REGION Network 15: IO evaluation — Instrument read and scale - Part 2
   // ▀▀▀▀▀▀▀▀▀▀▀▀▀▀▀▀▀▀▀▀▀▀▀▀▀▀▀▀▀▀▀▀▀▀▀▀▀▀▀▀▀▀▀▀
   // Scale value calculation part 2 (SCALE_MAX − SCALE_MIN)
   // ▄▄▄▄▄▄▄▄▄▄▄▄▄▄▄▄▄▄▄▄▄▄▄▄▄▄▄▄▄▄▄▄▄▄▄▄▄▄▄▄▄▄▄▄
   RUNG wire#powerrail
      { S7_Templates := "SrcType := Real"; S7_GenerateENO := "TRUE" } Sub(in1 := #STATIC_DATA.RANGE_SCALE_MAX, in2 := #STATIC_DATA.RANGE_SCALE_MIN, out => #calcPart2)
   END_RUNG
   // the same network as SCL:
   #calcPart2 := #STATIC_DATA.RANGE_SCALE_MAX - #STATIC_DATA.RANGE_SCALE_MIN;
END_REGION

REGION Network 16: IO evaluation — Instrument read and scale - Part 3
   // ▀▀▀▀▀▀▀▀▀▀▀▀▀▀▀▀▀▀▀▀▀▀▀▀▀▀▀▀▀▀▀▀▀▀▀▀▀▀▀▀▀▀▀▀
   // Scale value calculation part 3 (RAW_MAX − RAW_MIN)
   // 
   // Note:    To prevent inconsistencies and divide by zero errors, if a configuration error is present
   //      (resulting from incorrect range data and indicated by status_ConfigError = TRUE), the
   //      denominator of the calculation (CalcPart3) is set to 3.402823 × 1038 (i.e. a very large 
   //      number), the result of this is that the  actual_Value will equal RANGE_SCALE_MIN for 
   //      all permitted values of RAW_ANALOG.
   // ▄▄▄▄▄▄▄▄▄▄▄▄▄▄▄▄▄▄▄▄▄▄▄▄▄▄▄▄▄▄▄▄▄▄▄▄▄▄▄▄▄▄▄▄
   RUNG wire#powerrail
      { S7_Templates := "SrcType := Real"; S7_GenerateENO := "TRUE" } Sub(in1 := #STATIC_DATA.RANGE_RAW_MAX, in2 := #STATIC_DATA.RANGE_RAW_MIN, out => #calcPart3)
      Contact( #DYNAMIC_DATA.status_ConfigError )
      Move(in := 3.402823E+38, out1 => #calcPart3)
   END_RUNG
   // the same network as SCL:
   // ENO of a box is taken as its EN; it also drops when the box reports an error
   #calcPart3 := #STATIC_DATA.RANGE_RAW_MAX - #STATIC_DATA.RANGE_RAW_MIN;
   IF #DYNAMIC_DATA.status_ConfigError THEN #calcPart3 := 3.402823E+38; END_IF;
END_REGION

REGION Network 17: IO evaluation — Instrument read and scale - Part 4
   // ▀▀▀▀▀▀▀▀▀▀▀▀▀▀▀▀▀▀▀▀▀▀▀▀▀▀▀▀▀▀▀▀▀▀▀▀▀▀▀▀▀▀▀▀
   //                                                                              (calcPart1 x CalcPart2)
   // Complete the calculation SCALE_VALUE =  —————————— + SCALE_MIN
   //                                                                                         calcPart3
   // 
   // If a configuration error exists, the actual value is set to zero for all conditions
   // ▄▄▄▄▄▄▄▄▄▄▄▄▄▄▄▄▄▄▄▄▄▄▄▄▄▄▄▄▄▄▄▄▄▄▄▄▄▄▄▄▄▄▄▄
   RUNG wire#powerrail
      { S7_Templates := "SrcType := Real"; S7_GenerateENO := "TRUE" } Mul(in1 := #calcPart1, in2 := #calcPart2, out => #wrkReal)
      { S7_Templates := "SrcType := Real"; S7_GenerateENO := "TRUE" } Div(in1 := #wrkReal, in2 := #calcPart3, out => #wrkReal)
      { S7_Templates := "SrcType := Real"; S7_GenerateENO := "TRUE" } Add(in1 := #wrkReal, in2 := #STATIC_DATA.RANGE_SCALE_MIN, out => #DYNAMIC_DATA.actual_Value)
   END_RUNG
   RUNG wire#powerrail
      Contact( #DYNAMIC_DATA.status_ConfigError )
      Move(in := 0.0, out1 => #DYNAMIC_DATA.actual_Value)
   END_RUNG
   // the same network as SCL:
   // ENO of a box is taken as its EN; it also drops when the box reports an error
   #wrkReal := #calcPart1 * #calcPart2;
   #wrkReal := #wrkReal / #calcPart3;
   #DYNAMIC_DATA.actual_Value := #wrkReal + #STATIC_DATA.RANGE_SCALE_MIN;
   IF #DYNAMIC_DATA.status_ConfigError THEN #DYNAMIC_DATA.actual_Value := 0.0; END_IF;
END_REGION

REGION Network 18: IO evaluation — Calculate out of range value
   // ▀▀▀▀▀▀▀▀▀▀▀▀▀▀▀▀▀▀▀▀▀▀▀▀▀▀▀▀▀▀▀▀▀▀▀▀▀▀▀▀▀▀▀▀
   // The out of range limits are calculated from the raw span of the instrument 
   // (RAW_MAX - RAW_MIN, stored in calcPart3).
   // 
   // The absolute value of the out of range tolerance is stored in calcRawOOR and is calculated as
   // follows:
   // 
   // 
   //                                (RAW_MAX - RAW_MIN) x wrkOORPercent
   // calcRawOOR  =  ————————————————————
   //                                                                100
   // 
   // OR
   // 
   //                               calcPart3 x wrkOORPercent
   // calcRawOOR  =  ——————————————
   //                                                 100
   // 
   // 
   // The instrument is over range if the RAW_ANALOG is greater than RAW_MAX + calcRawOOR
   // 
   // The instrument is under range if the RAW_ANALOG is less than RAW_MIN - calcRawOOR
   // ▄▄▄▄▄▄▄▄▄▄▄▄▄▄▄▄▄▄▄▄▄▄▄▄▄▄▄▄▄▄▄▄▄▄▄▄▄▄▄▄▄▄▄▄
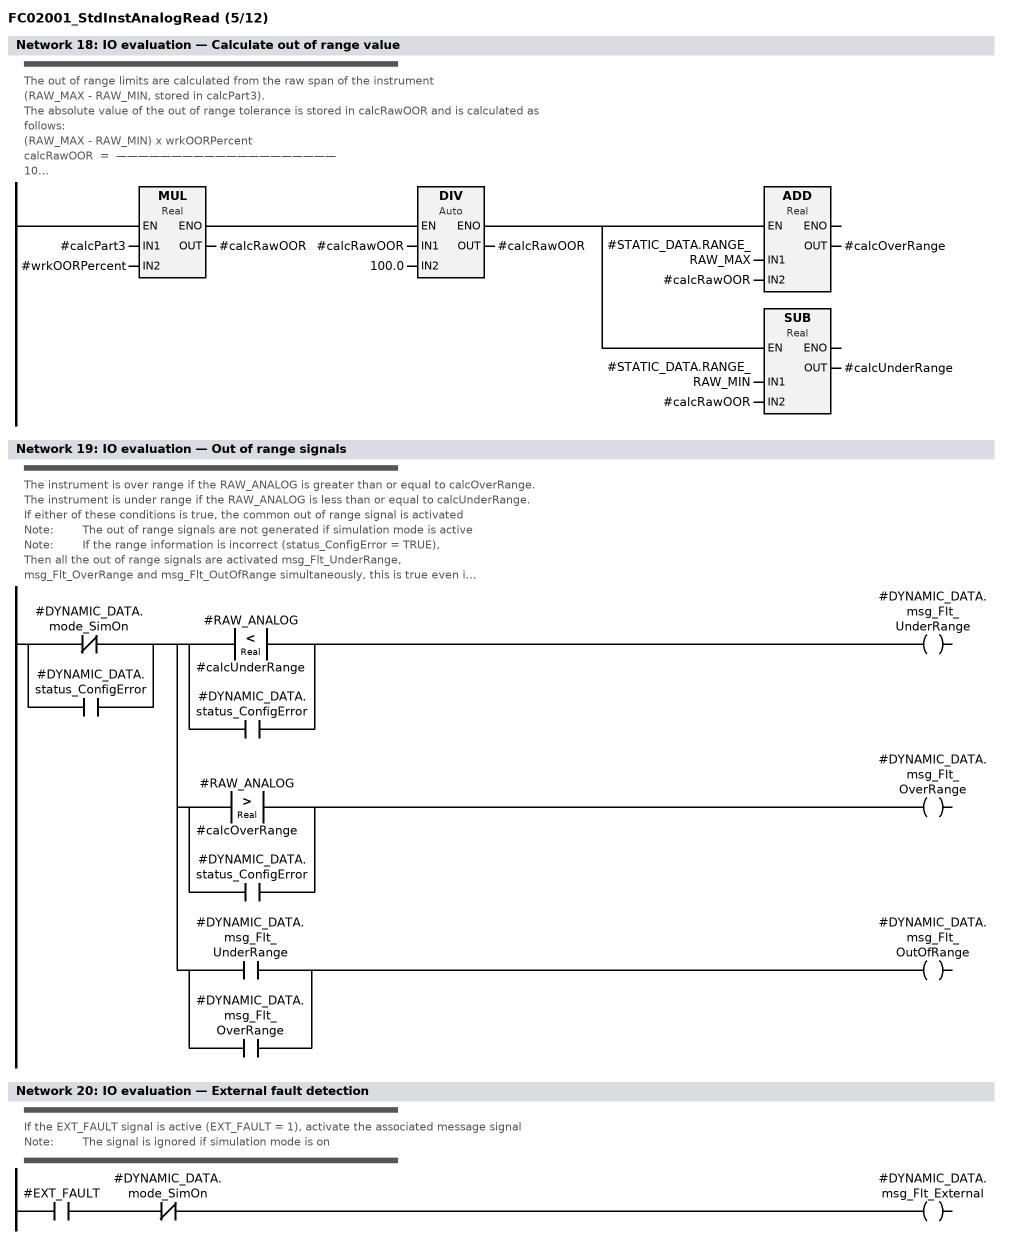
   RUNG wire#powerrail
      { S7_Templates := "SrcType := Real"; S7_GenerateENO := "TRUE" } Mul(in1 := #calcPart3, in2 := #wrkOORPercent, out => #calcRawOOR)
      Div(in1 := #calcRawOOR, in2 := 100.0, out => #calcRawOOR)
      wire#w1
      { S7_Templates := "SrcType := Real"; S7_GenerateENO := "TRUE" } Add(in1 := #STATIC_DATA.RANGE_RAW_MAX, in2 := #calcRawOOR, out => #calcOverRange)
   END_RUNG
   RUNG wire#w1
      { S7_Templates := "SrcType := Real"; S7_GenerateENO := "TRUE" } Sub(in1 := #STATIC_DATA.RANGE_RAW_MIN, in2 := #calcRawOOR, out => #calcUnderRange)
   END_RUNG
   // the same network as SCL:
   // ENO of a box is taken as its EN; it also drops when the box reports an error
   #calcRawOOR := #calcPart3 * #wrkOORPercent;
   #calcRawOOR := #calcRawOOR / 100.0;
   #calcOverRange := #STATIC_DATA.RANGE_RAW_MAX + #calcRawOOR;
   #calcUnderRange := #STATIC_DATA.RANGE_RAW_MIN - #calcRawOOR;
END_REGION

REGION Network 19: IO evaluation — Out of range signals
   // ▀▀▀▀▀▀▀▀▀▀▀▀▀▀▀▀▀▀▀▀▀▀▀▀▀▀▀▀▀▀▀▀▀▀▀▀▀▀▀▀▀▀▀▀
   // The instrument is over range if the RAW_ANALOG is greater than or equal to calcOverRange.
   // 
   // The instrument is under range if the RAW_ANALOG is less than or equal to calcUnderRange.
   // 
   // If either of these conditions is true, the common out of range signal is activated
   // 
   // Note:    The out of range signals are not generated if simulation mode is active
   // 
   // Note:    If the range information is incorrect (status_ConfigError = TRUE),
   //      Then all the out of range signals are activated msg_Flt_UnderRange, 
   //      msg_Flt_OverRange and msg_Flt_OutOfRange simultaneously, this is true even if
   //      simulation mode is active.
   // ▄▄▄▄▄▄▄▄▄▄▄▄▄▄▄▄▄▄▄▄▄▄▄▄▄▄▄▄▄▄▄▄▄▄▄▄▄▄▄▄▄▄▄▄
   RUNG wire#powerrail
      I_Contact( #DYNAMIC_DATA.mode_SimOn )
      wire#w1
      { S7_Templates := "SrcType := Real" } LT_Contact(in1 := #RAW_ANALOG, in2 := #calcUnderRange)
      wire#w2
      Coil( #DYNAMIC_DATA.msg_Flt_UnderRange )
   END_RUNG
   RUNG wire#powerrail
      Contact( #DYNAMIC_DATA.status_ConfigError )
   END_RUNG wire#w1
   RUNG wire#w1
      Contact( #DYNAMIC_DATA.status_ConfigError )
   END_RUNG wire#w2
   RUNG wire#w1
      { S7_Templates := "SrcType := Real" } GT_Contact(in1 := #RAW_ANALOG, in2 := #calcOverRange)
      wire#w3
      Coil( #DYNAMIC_DATA.msg_Flt_OverRange )
   END_RUNG
   RUNG wire#w1
      Contact( #DYNAMIC_DATA.status_ConfigError )
   END_RUNG wire#w3
   RUNG wire#w1
      Contact( #DYNAMIC_DATA.msg_Flt_UnderRange )
      wire#w4
      Coil( #DYNAMIC_DATA.msg_Flt_OutOfRange )
   END_RUNG
   RUNG wire#w1
      Contact( #DYNAMIC_DATA.msg_Flt_OverRange )
   END_RUNG wire#w4
   // the same network as SCL:
   #_w1 := NOT #DYNAMIC_DATA.mode_SimOn OR #DYNAMIC_DATA.status_ConfigError;
   #DYNAMIC_DATA.msg_Flt_UnderRange := #_w1 AND ((#RAW_ANALOG < #calcUnderRange) OR #DYNAMIC_DATA.status_ConfigError);
   #DYNAMIC_DATA.msg_Flt_OverRange := #_w1 AND ((#RAW_ANALOG > #calcOverRange) OR #DYNAMIC_DATA.status_ConfigError);
   #DYNAMIC_DATA.msg_Flt_OutOfRange := #_w1 AND (#DYNAMIC_DATA.msg_Flt_UnderRange OR #DYNAMIC_DATA.msg_Flt_OverRange);
END_REGION

REGION Network 20: IO evaluation — External fault detection
   // ▀▀▀▀▀▀▀▀▀▀▀▀▀▀▀▀▀▀▀▀▀▀▀▀▀▀▀▀▀▀▀▀▀▀▀▀▀▀▀▀▀▀▀▀
   // If the EXT_FAULT signal is active (EXT_FAULT = 1), activate the associated message signal
   // 
   // Note:    The signal is ignored if simulation mode is on
   // ▄▄▄▄▄▄▄▄▄▄▄▄▄▄▄▄▄▄▄▄▄▄▄▄▄▄▄▄▄▄▄▄▄▄▄▄▄▄▄▄▄▄▄▄
   RUNG wire#powerrail
      Contact( #EXT_FAULT )
      I_Contact( #DYNAMIC_DATA.mode_SimOn )
      Coil( #DYNAMIC_DATA.msg_Flt_External )
   END_RUNG
   // the same network as SCL:
   #DYNAMIC_DATA.msg_Flt_External := #EXT_FAULT AND NOT #DYNAMIC_DATA.mode_SimOn;
END_REGION

REGION Network 21: Operating mode — Simulation mode
   // ▀▀▀▀▀▀▀▀▀▀▀▀▀▀▀▀▀▀▀▀▀▀▀▀▀▀▀▀▀▀▀▀▀▀▀▀▀▀▀▀▀▀▀▀
   // If simulation mode is enabled (mode_SimOn = 1) and a configuration error is not present,
   // (status_ConfigError = 0) overwrite the actual_Value with the mode_SimValue signal set by the 
   // operator.
   // 
   // Note:    Any fault signals will be suppressed (turned off) is simulation mode is active
   //      and a configuration error is not present
   // 
   //      The simulated value (mode_SimValue) is restricted to the range given in 
   //      RANGE_SCALE_MIN and RANGE_SCALE_MAX
   // ▄▄▄▄▄▄▄▄▄▄▄▄▄▄▄▄▄▄▄▄▄▄▄▄▄▄▄▄▄▄▄▄▄▄▄▄▄▄▄▄▄▄▄▄
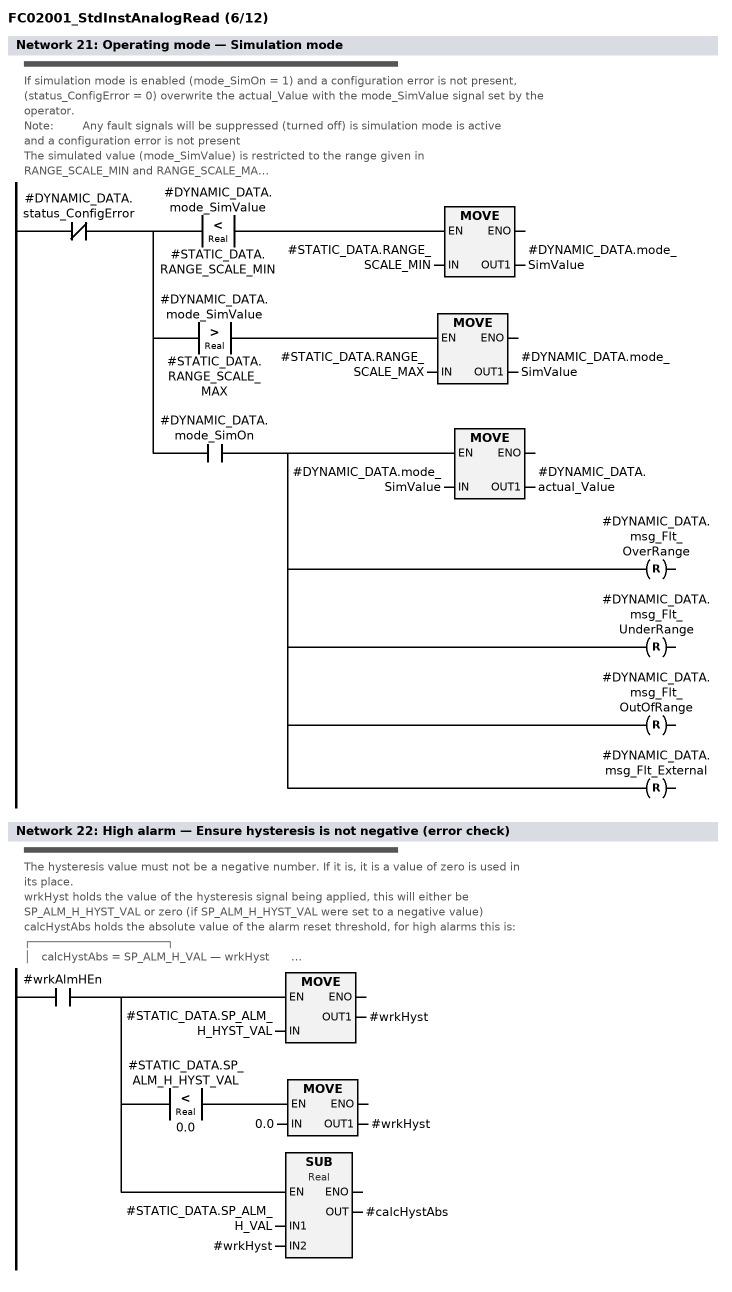
   RUNG wire#powerrail
      I_Contact( #DYNAMIC_DATA.status_ConfigError )
      wire#w1
      { S7_Templates := "SrcType := Real" } LT_Contact(in1 := #DYNAMIC_DATA.mode_SimValue, in2 := #STATIC_DATA.RANGE_SCALE_MIN)
      { S7_GenerateENO := "TRUE" } Move(in := #STATIC_DATA.RANGE_SCALE_MIN, out1 => #DYNAMIC_DATA.mode_SimValue)
   END_RUNG
   RUNG wire#w1
      { S7_Templates := "SrcType := Real" } GT_Contact(in1 := #DYNAMIC_DATA.mode_SimValue, in2 := #STATIC_DATA.RANGE_SCALE_MAX)
      { S7_GenerateENO := "TRUE" } Move(in := #STATIC_DATA.RANGE_SCALE_MAX, out1 => #DYNAMIC_DATA.mode_SimValue)
   END_RUNG
   RUNG wire#w1
      Contact( #DYNAMIC_DATA.mode_SimOn )
      wire#w2
      { S7_GenerateENO := "TRUE" } Move(in := #DYNAMIC_DATA.mode_SimValue, out1 => #DYNAMIC_DATA.actual_Value)
   END_RUNG
   RUNG wire#w2
      R_Coil( #DYNAMIC_DATA.msg_Flt_OverRange )
   END_RUNG
   RUNG wire#w2
      R_Coil( #DYNAMIC_DATA.msg_Flt_UnderRange )
   END_RUNG
   RUNG wire#w2
      R_Coil( #DYNAMIC_DATA.msg_Flt_OutOfRange )
   END_RUNG
   RUNG wire#w2
      R_Coil( #DYNAMIC_DATA.msg_Flt_External )
   END_RUNG
   // the same network as SCL:
   #_w1 := NOT #DYNAMIC_DATA.status_ConfigError;
   IF #_w1 AND (#DYNAMIC_DATA.mode_SimValue < #STATIC_DATA.RANGE_SCALE_MIN) THEN
       #DYNAMIC_DATA.mode_SimValue := #STATIC_DATA.RANGE_SCALE_MIN;
   END_IF;
   IF #_w1 AND (#DYNAMIC_DATA.mode_SimValue > #STATIC_DATA.RANGE_SCALE_MAX) THEN
       #DYNAMIC_DATA.mode_SimValue := #STATIC_DATA.RANGE_SCALE_MAX;
   END_IF;
   IF #_w1 AND #DYNAMIC_DATA.mode_SimOn THEN
       #DYNAMIC_DATA.actual_Value := #DYNAMIC_DATA.mode_SimValue;
       #DYNAMIC_DATA.msg_Flt_OverRange := FALSE;
       #DYNAMIC_DATA.msg_Flt_UnderRange := FALSE;
       #DYNAMIC_DATA.msg_Flt_OutOfRange := FALSE;
       #DYNAMIC_DATA.msg_Flt_External := FALSE;
   END_IF;
END_REGION

REGION Network 22: High alarm — Ensure hysteresis is not negative (error check)
   // ▀▀▀▀▀▀▀▀▀▀▀▀▀▀▀▀▀▀▀▀▀▀▀▀▀▀▀▀▀▀▀▀▀▀▀▀▀▀▀▀▀▀▀▀
   // The hysteresis value must not be a negative number. If it is, it is a value of zero is used in
   // its place.
   // 
   // wrkHyst holds the value of the hysteresis signal being applied, this will either be 
   // SP_ALM_H_HYST_VAL or zero (if SP_ALM_H_HYST_VAL were set to a negative value)
   // 
   // calcHystAbs holds the absolute value of the alarm reset threshold, for high alarms this is:
   // ┌─────────────────────┐
   // │ calcHystAbs = SP_ALM_H_VAL — wrkHyst    │
   // └─────────────────────┘
   // 
   // The two threshold values for the high alarm are thus:
   // 
   //      High alarm activation threshold = SP_ALM_H_VAL
   //      High alarm reset threshold          = calcHystAbs
   // 
   // Note:    The hysteresis is only checked if alarm is being evaluated
   // ▄▄▄▄▄▄▄▄▄▄▄▄▄▄▄▄▄▄▄▄▄▄▄▄▄▄▄▄▄▄▄▄▄▄▄▄▄▄▄▄▄▄▄▄
   RUNG wire#powerrail
      Contact( #wrkAlmHEn )
      wire#w1
      { S7_GenerateENO := "TRUE" } Move(in := #STATIC_DATA.SP_ALM_H_HYST_VAL, out1 => #wrkHyst)
   END_RUNG
   RUNG wire#w1
      { S7_Templates := "SrcType := Real" } LT_Contact(in1 := #STATIC_DATA.SP_ALM_H_HYST_VAL, in2 := 0.0)
      { S7_GenerateENO := "TRUE" } Move(in := 0.0, out1 => #wrkHyst)
   END_RUNG
   RUNG wire#w1
      { S7_Templates := "SrcType := Real"; S7_GenerateENO := "TRUE" } Sub(in1 := #STATIC_DATA.SP_ALM_H_VAL, in2 := #wrkHyst, out => #calcHystAbs)
   END_RUNG
   // the same network as SCL:
   IF #wrkAlmHEn THEN #wrkHyst := #STATIC_DATA.SP_ALM_H_HYST_VAL; END_IF;
   IF #wrkAlmHEn AND (#STATIC_DATA.SP_ALM_H_HYST_VAL < 0.0) THEN #wrkHyst := 0.0; END_IF;
   IF #wrkAlmHEn THEN #calcHystAbs := #STATIC_DATA.SP_ALM_H_VAL - #wrkHyst; END_IF;
END_REGION

REGION Network 23: High alarm — Check for activation level and ON-DELAY timer
   // ▀▀▀▀▀▀▀▀▀▀▀▀▀▀▀▀▀▀▀▀▀▀▀▀▀▀▀▀▀▀▀▀▀▀▀▀▀▀▀▀▀▀▀▀
   // If the high alarm has been enabled and is not masked and the actual_Value is greater than or 
   // equal to the alarm setpoint (SP_ALM_H_VAL), but the alarm has not yet been triggered 
   // (msg_Alm_H = 0) then the ON-DELAY phase is active (the alarm timer is counting down).
   // 
   // The timer will begin to count down from the value in TIME_ALM_H_ON_DEL using the 200ms 
   // pulse (it will count down in increments of 0.2s). If the high alarm timer is less than or equal to 
   // zero, then the ON-DELAY has expired and the High Alarm message will become active.
   // 
   // If at any point during the ON-DELAY count down, the actual_Value drops below the activation
   // setpoint (SP_ALM_H_VAL), the timer will be reset to the TIME_ALM_H_ON_DEL value, forcing 
   // the ON-DELAY to start again.
   // ▄▄▄▄▄▄▄▄▄▄▄▄▄▄▄▄▄▄▄▄▄▄▄▄▄▄▄▄▄▄▄▄▄▄▄▄▄▄▄▄▄▄▄▄
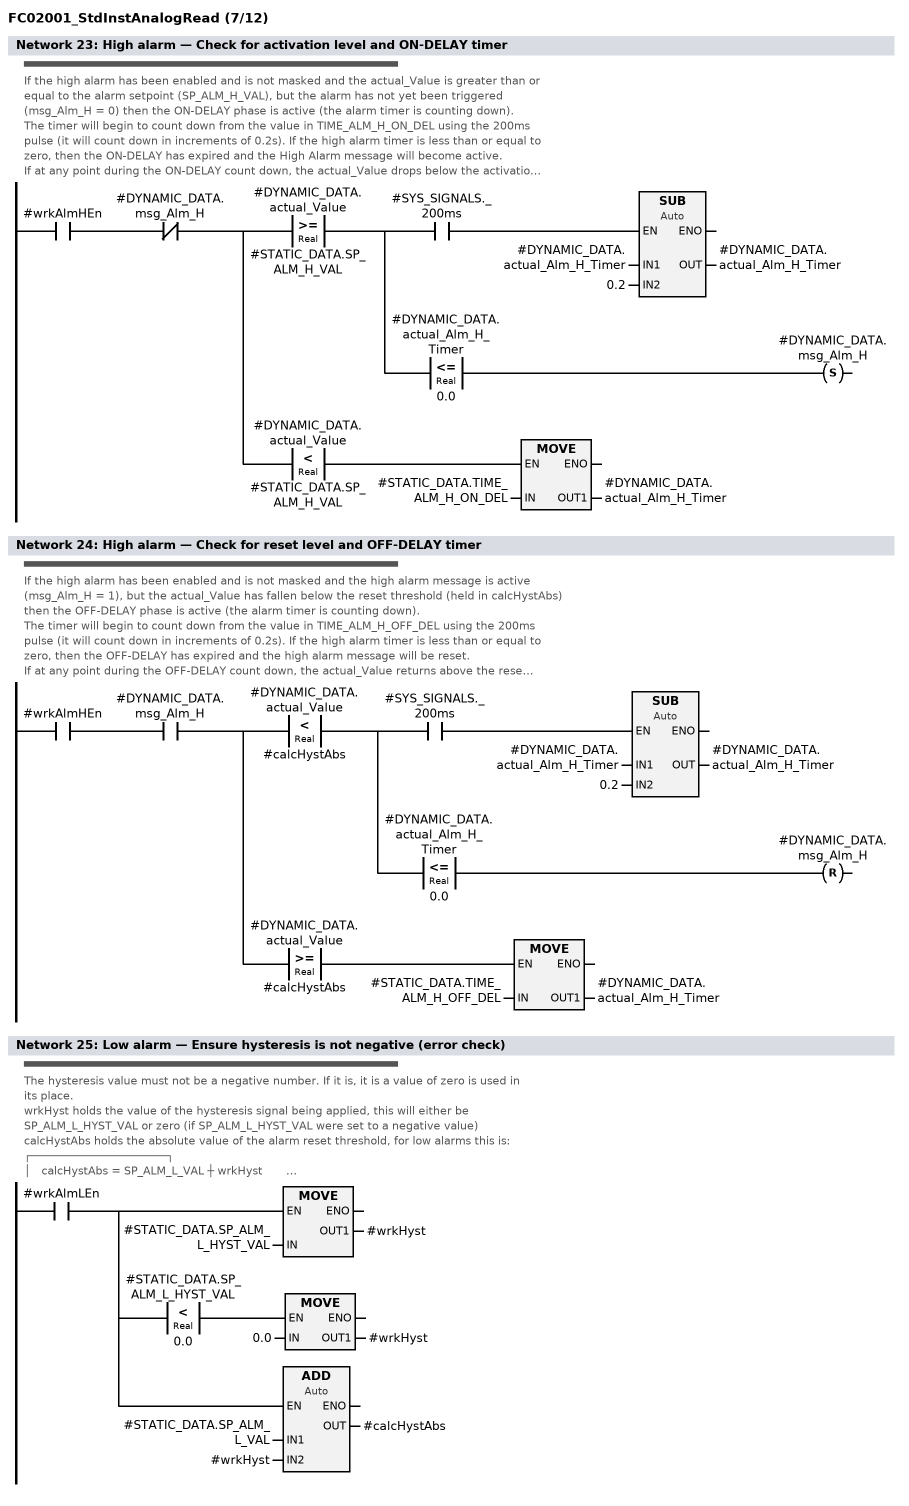
   RUNG wire#powerrail
      Contact( #wrkAlmHEn )
      I_Contact( #DYNAMIC_DATA.msg_Alm_H )
      wire#w1
      { S7_Templates := "SrcType := Real" } GE_Contact(in1 := #DYNAMIC_DATA.actual_Value, in2 := #STATIC_DATA.SP_ALM_H_VAL)
      wire#w2
      Contact( #SYS_SIGNALS._200ms )
      Sub(in1 := #DYNAMIC_DATA.actual_Alm_H_Timer, in2 := 0.2, out => #DYNAMIC_DATA.actual_Alm_H_Timer)
   END_RUNG
   RUNG wire#w2
      { S7_Templates := "SrcType := Real" } LE_Contact(in1 := #DYNAMIC_DATA.actual_Alm_H_Timer, in2 := 0.0)
      S_Coil( #DYNAMIC_DATA.msg_Alm_H )
   END_RUNG
   RUNG wire#w1
      { S7_Templates := "SrcType := Real" } LT_Contact(in1 := #DYNAMIC_DATA.actual_Value, in2 := #STATIC_DATA.SP_ALM_H_VAL)
      { S7_GenerateENO := "TRUE" } Move(in := #STATIC_DATA.TIME_ALM_H_ON_DEL, out1 => #DYNAMIC_DATA.actual_Alm_H_Timer)
   END_RUNG
   // the same network as SCL:
   #_w1 := #wrkAlmHEn AND NOT #DYNAMIC_DATA.msg_Alm_H;
   #_w2 := #_w1 AND (#DYNAMIC_DATA.actual_Value >= #STATIC_DATA.SP_ALM_H_VAL);
   IF #_w2 AND #SYS_SIGNALS._200ms THEN
       #DYNAMIC_DATA.actual_Alm_H_Timer := #DYNAMIC_DATA.actual_Alm_H_Timer - 0.2;
   END_IF;
   IF #_w2 AND (#DYNAMIC_DATA.actual_Alm_H_Timer <= 0.0) THEN #DYNAMIC_DATA.msg_Alm_H := TRUE; END_IF;
   IF #_w1 AND (#DYNAMIC_DATA.actual_Value < #STATIC_DATA.SP_ALM_H_VAL) THEN
       #DYNAMIC_DATA.actual_Alm_H_Timer := #STATIC_DATA.TIME_ALM_H_ON_DEL;
   END_IF;
END_REGION

REGION Network 24: High alarm — Check for reset level and OFF-DELAY timer
   // ▀▀▀▀▀▀▀▀▀▀▀▀▀▀▀▀▀▀▀▀▀▀▀▀▀▀▀▀▀▀▀▀▀▀▀▀▀▀▀▀▀▀▀▀
   // If the high alarm has been enabled and is not masked and the high alarm message is active 
   // (msg_Alm_H = 1), but the actual_Value has fallen below the reset threshold (held in calcHystAbs) 
   // then the OFF-DELAY phase is active (the alarm timer is counting down).
   // 
   // The timer will begin to count down from the value in TIME_ALM_H_OFF_DEL using the 200ms 
   // pulse (it will count down in increments of 0.2s). If the high alarm timer is less than or equal to 
   // zero, then the OFF-DELAY has expired and the high alarm message will be reset.
   // 
   // If at any point during the OFF-DELAY count down, the actual_Value returns above the reset
   // threshold (calcHystAbs), the timer will be reset to the TIME_ALM_H_OFF_DEL value, forcing 
   // the OFF-DELAY to start again.
   // ▄▄▄▄▄▄▄▄▄▄▄▄▄▄▄▄▄▄▄▄▄▄▄▄▄▄▄▄▄▄▄▄▄▄▄▄▄▄▄▄▄▄▄▄
   RUNG wire#powerrail
      Contact( #wrkAlmHEn )
      Contact( #DYNAMIC_DATA.msg_Alm_H )
      wire#w1
      { S7_Templates := "SrcType := Real" } LT_Contact(in1 := #DYNAMIC_DATA.actual_Value, in2 := #calcHystAbs)
      wire#w2
      Contact( #SYS_SIGNALS._200ms )
      Sub(in1 := #DYNAMIC_DATA.actual_Alm_H_Timer, in2 := 0.2, out => #DYNAMIC_DATA.actual_Alm_H_Timer)
   END_RUNG
   RUNG wire#w2
      { S7_Templates := "SrcType := Real" } LE_Contact(in1 := #DYNAMIC_DATA.actual_Alm_H_Timer, in2 := 0.0)
      R_Coil( #DYNAMIC_DATA.msg_Alm_H )
   END_RUNG
   RUNG wire#w1
      { S7_Templates := "SrcType := Real" } GE_Contact(in1 := #DYNAMIC_DATA.actual_Value, in2 := #calcHystAbs)
      { S7_GenerateENO := "TRUE" } Move(in := #STATIC_DATA.TIME_ALM_H_OFF_DEL, out1 => #DYNAMIC_DATA.actual_Alm_H_Timer)
   END_RUNG
   // the same network as SCL:
   #_w1 := #wrkAlmHEn AND #DYNAMIC_DATA.msg_Alm_H;
   #_w2 := #_w1 AND (#DYNAMIC_DATA.actual_Value < #calcHystAbs);
   IF #_w2 AND #SYS_SIGNALS._200ms THEN
       #DYNAMIC_DATA.actual_Alm_H_Timer := #DYNAMIC_DATA.actual_Alm_H_Timer - 0.2;
   END_IF;
   IF #_w2 AND (#DYNAMIC_DATA.actual_Alm_H_Timer <= 0.0) THEN #DYNAMIC_DATA.msg_Alm_H := FALSE; END_IF;
   IF #_w1 AND (#DYNAMIC_DATA.actual_Value >= #calcHystAbs) THEN
       #DYNAMIC_DATA.actual_Alm_H_Timer := #STATIC_DATA.TIME_ALM_H_OFF_DEL;
   END_IF;
END_REGION

REGION Network 25: Low alarm — Ensure hysteresis is not negative (error check)
   // ▀▀▀▀▀▀▀▀▀▀▀▀▀▀▀▀▀▀▀▀▀▀▀▀▀▀▀▀▀▀▀▀▀▀▀▀▀▀▀▀▀▀▀▀
   // The hysteresis value must not be a negative number. If it is, it is a value of zero is used in
   // its place.
   // 
   // wrkHyst holds the value of the hysteresis signal being applied, this will either be 
   // SP_ALM_L_HYST_VAL or zero (if SP_ALM_L_HYST_VAL were set to a negative value)
   // 
   // calcHystAbs holds the absolute value of the alarm reset threshold, for low alarms this is:
   // ┌─────────────────────┐
   // │ calcHystAbs = SP_ALM_L_VAL ┼ wrkHyst     │
   // └─────────────────────┘
   // 
   // The two threshold values for the low alarm are thus:
   // 
   //      Low alarm activation threshold = SP_ALM_L_VAL
   //      Low alarm reset threshold          = calcHystAbs
   // 
   // Note:    The hysteresis is only checked if alarm is being evaluated
   // ▄▄▄▄▄▄▄▄▄▄▄▄▄▄▄▄▄▄▄▄▄▄▄▄▄▄▄▄▄▄▄▄▄▄▄▄▄▄▄▄▄▄▄▄
   RUNG wire#powerrail
      Contact( #wrkAlmLEn )
      wire#w1
      { S7_GenerateENO := "TRUE" } Move(in := #STATIC_DATA.SP_ALM_L_HYST_VAL, out1 => #wrkHyst)
   END_RUNG
   RUNG wire#w1
      { S7_Templates := "SrcType := Real" } LT_Contact(in1 := #STATIC_DATA.SP_ALM_L_HYST_VAL, in2 := 0.0)
      { S7_GenerateENO := "TRUE" } Move(in := 0.0, out1 => #wrkHyst)
   END_RUNG
   RUNG wire#w1
      Add(in1 := #STATIC_DATA.SP_ALM_L_VAL, in2 := #wrkHyst, out => #calcHystAbs)
   END_RUNG
   // the same network as SCL:
   IF #wrkAlmLEn THEN #wrkHyst := #STATIC_DATA.SP_ALM_L_HYST_VAL; END_IF;
   IF #wrkAlmLEn AND (#STATIC_DATA.SP_ALM_L_HYST_VAL < 0.0) THEN #wrkHyst := 0.0; END_IF;
   IF #wrkAlmLEn THEN #calcHystAbs := #STATIC_DATA.SP_ALM_L_VAL + #wrkHyst; END_IF;
END_REGION

REGION Network 26: Low alarm — Check for activation level and ON-DELAY timer
   // ▀▀▀▀▀▀▀▀▀▀▀▀▀▀▀▀▀▀▀▀▀▀▀▀▀▀▀▀▀▀▀▀▀▀▀▀▀▀▀▀▀▀▀▀
   // If the low alarm has been enabled and is not masked and the actual_Value is less than or 
   // equal to the alarm setpoint (SP_ALM_L_VAL), but the alarm has not yet been triggered 
   // (msg_Alm_L = 0) then the ON-DELAY phase is active (the alarm timer is counting down).
   // 
   // The timer will begin to count down from the value in TIME_ALM_L_ON_DEL using the 200ms 
   // pulse (it will count down in increments of 0.2s). If the Low alarm timer is less than or equal to 
   // zero, then the ON-DELAY has expired and the Low Alarm message will become active.
   // 
   // If at any point during the ON-DELAY count down, the actual_Value rises above the activation
   // setpoint (SP_ALM_L_VAL), the timer will be reset to the TIME_ALM_L_ON_DEL value, forcing 
   // the ON-DELAY to start again.
   // ▄▄▄▄▄▄▄▄▄▄▄▄▄▄▄▄▄▄▄▄▄▄▄▄▄▄▄▄▄▄▄▄▄▄▄▄▄▄▄▄▄▄▄▄
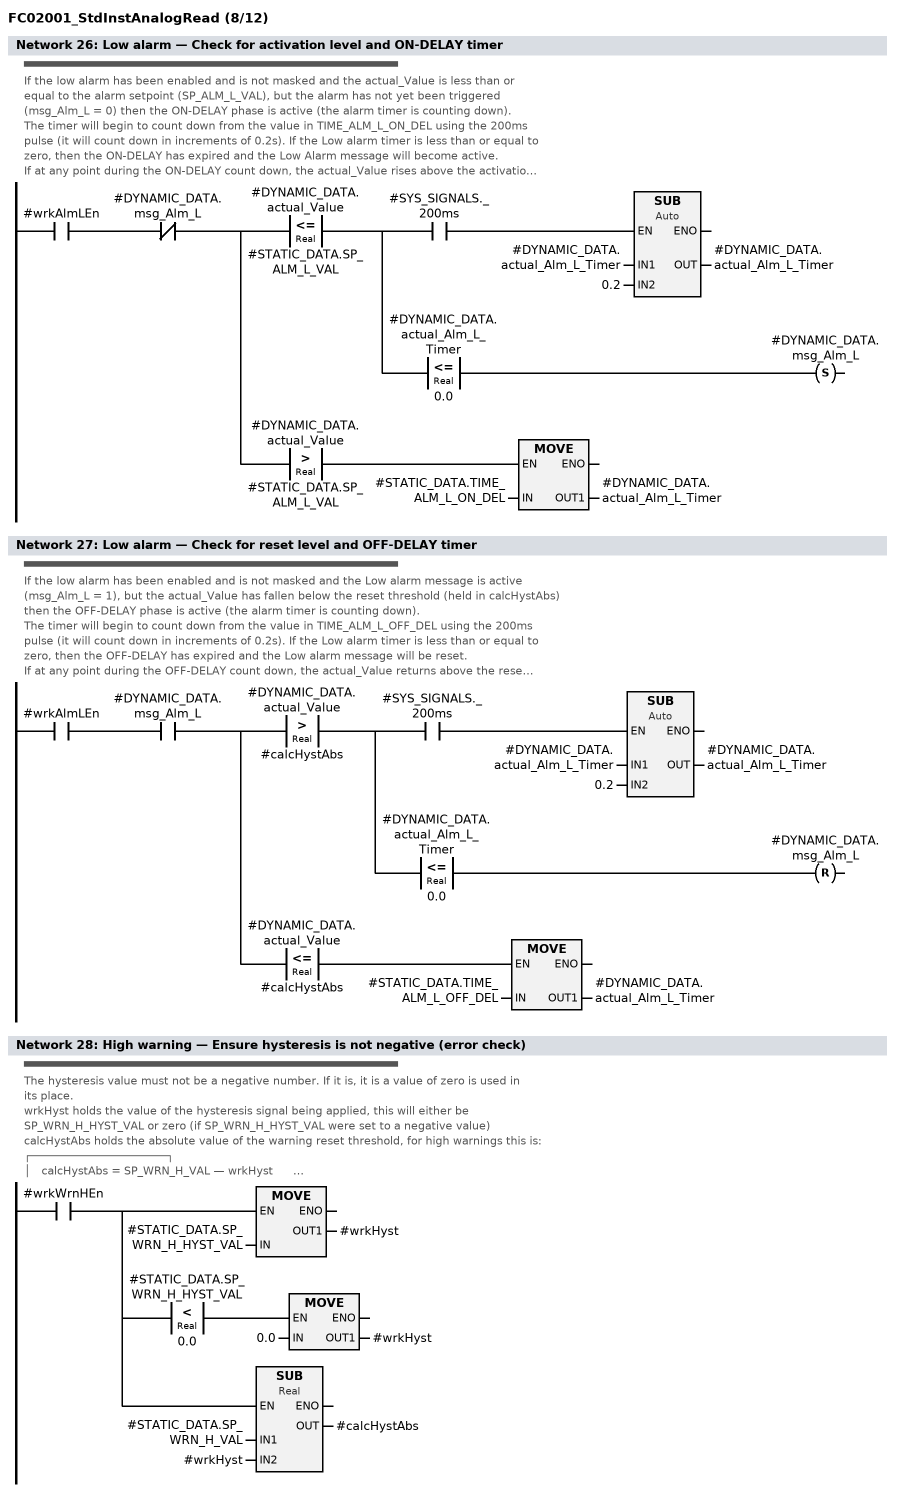
   RUNG wire#powerrail
      Contact( #wrkAlmLEn )
      I_Contact( #DYNAMIC_DATA.msg_Alm_L )
      wire#w1
      { S7_Templates := "SrcType := Real" } LE_Contact(in1 := #DYNAMIC_DATA.actual_Value, in2 := #STATIC_DATA.SP_ALM_L_VAL)
      wire#w2
      Contact( #SYS_SIGNALS._200ms )
      Sub(in1 := #DYNAMIC_DATA.actual_Alm_L_Timer, in2 := 0.2, out => #DYNAMIC_DATA.actual_Alm_L_Timer)
   END_RUNG
   RUNG wire#w2
      { S7_Templates := "SrcType := Real" } LE_Contact(in1 := #DYNAMIC_DATA.actual_Alm_L_Timer, in2 := 0.0)
      S_Coil( #DYNAMIC_DATA.msg_Alm_L )
   END_RUNG
   RUNG wire#w1
      { S7_Templates := "SrcType := Real" } GT_Contact(in1 := #DYNAMIC_DATA.actual_Value, in2 := #STATIC_DATA.SP_ALM_L_VAL)
      { S7_GenerateENO := "TRUE" } Move(in := #STATIC_DATA.TIME_ALM_L_ON_DEL, out1 => #DYNAMIC_DATA.actual_Alm_L_Timer)
   END_RUNG
   // the same network as SCL:
   #_w1 := #wrkAlmLEn AND NOT #DYNAMIC_DATA.msg_Alm_L;
   #_w2 := #_w1 AND (#DYNAMIC_DATA.actual_Value <= #STATIC_DATA.SP_ALM_L_VAL);
   IF #_w2 AND #SYS_SIGNALS._200ms THEN
       #DYNAMIC_DATA.actual_Alm_L_Timer := #DYNAMIC_DATA.actual_Alm_L_Timer - 0.2;
   END_IF;
   IF #_w2 AND (#DYNAMIC_DATA.actual_Alm_L_Timer <= 0.0) THEN #DYNAMIC_DATA.msg_Alm_L := TRUE; END_IF;
   IF #_w1 AND (#DYNAMIC_DATA.actual_Value > #STATIC_DATA.SP_ALM_L_VAL) THEN
       #DYNAMIC_DATA.actual_Alm_L_Timer := #STATIC_DATA.TIME_ALM_L_ON_DEL;
   END_IF;
END_REGION

REGION Network 27: Low alarm — Check for reset level and OFF-DELAY timer
   // ▀▀▀▀▀▀▀▀▀▀▀▀▀▀▀▀▀▀▀▀▀▀▀▀▀▀▀▀▀▀▀▀▀▀▀▀▀▀▀▀▀▀▀▀
   // If the low alarm has been enabled and is not masked and the Low alarm message is active 
   // (msg_Alm_L = 1), but the actual_Value has fallen below the reset threshold (held in calcHystAbs) 
   // then the OFF-DELAY phase is active (the alarm timer is counting down).
   // 
   // The timer will begin to count down from the value in TIME_ALM_L_OFF_DEL using the 200ms 
   // pulse (it will count down in increments of 0.2s). If the Low alarm timer is less than or equal to 
   // zero, then the OFF-DELAY has expired and the Low alarm message will be reset.
   // 
   // If at any point during the OFF-DELAY count down, the actual_Value returns above the reset
   // threshold (calcHystAbs), the timer will be reset to the TIME_ALM_L_OFF_DEL value, forcing 
   // the OFF-DELAY to start again.
   // ▄▄▄▄▄▄▄▄▄▄▄▄▄▄▄▄▄▄▄▄▄▄▄▄▄▄▄▄▄▄▄▄▄▄▄▄▄▄▄▄▄▄▄▄
   RUNG wire#powerrail
      Contact( #wrkAlmLEn )
      Contact( #DYNAMIC_DATA.msg_Alm_L )
      wire#w1
      { S7_Templates := "SrcType := Real" } GT_Contact(in1 := #DYNAMIC_DATA.actual_Value, in2 := #calcHystAbs)
      wire#w2
      Contact( #SYS_SIGNALS._200ms )
      Sub(in1 := #DYNAMIC_DATA.actual_Alm_L_Timer, in2 := 0.2, out => #DYNAMIC_DATA.actual_Alm_L_Timer)
   END_RUNG
   RUNG wire#w2
      { S7_Templates := "SrcType := Real" } LE_Contact(in1 := #DYNAMIC_DATA.actual_Alm_L_Timer, in2 := 0.0)
      R_Coil( #DYNAMIC_DATA.msg_Alm_L )
   END_RUNG
   RUNG wire#w1
      { S7_Templates := "SrcType := Real" } LE_Contact(in1 := #DYNAMIC_DATA.actual_Value, in2 := #calcHystAbs)
      { S7_GenerateENO := "TRUE" } Move(in := #STATIC_DATA.TIME_ALM_L_OFF_DEL, out1 => #DYNAMIC_DATA.actual_Alm_L_Timer)
   END_RUNG
   // the same network as SCL:
   #_w1 := #wrkAlmLEn AND #DYNAMIC_DATA.msg_Alm_L;
   #_w2 := #_w1 AND (#DYNAMIC_DATA.actual_Value > #calcHystAbs);
   IF #_w2 AND #SYS_SIGNALS._200ms THEN
       #DYNAMIC_DATA.actual_Alm_L_Timer := #DYNAMIC_DATA.actual_Alm_L_Timer - 0.2;
   END_IF;
   IF #_w2 AND (#DYNAMIC_DATA.actual_Alm_L_Timer <= 0.0) THEN #DYNAMIC_DATA.msg_Alm_L := FALSE; END_IF;
   IF #_w1 AND (#DYNAMIC_DATA.actual_Value <= #calcHystAbs) THEN
       #DYNAMIC_DATA.actual_Alm_L_Timer := #STATIC_DATA.TIME_ALM_L_OFF_DEL;
   END_IF;
END_REGION

REGION Network 28: High warning — Ensure hysteresis is not negative (error check)
   // ▀▀▀▀▀▀▀▀▀▀▀▀▀▀▀▀▀▀▀▀▀▀▀▀▀▀▀▀▀▀▀▀▀▀▀▀▀▀▀▀▀▀▀▀
   // The hysteresis value must not be a negative number. If it is, it is a value of zero is used in
   // its place.
   // 
   // wrkHyst holds the value of the hysteresis signal being applied, this will either be 
   // SP_WRN_H_HYST_VAL or zero (if SP_WRN_H_HYST_VAL were set to a negative value)
   // 
   // calcHystAbs holds the absolute value of the warning reset threshold, for high warnings this is:
   // ┌─────────────────────┐
   // │ calcHystAbs = SP_WRN_H_VAL — wrkHyst    │
   // └─────────────────────┘
   // 
   // The two threshold values for the high warning are thus:
   // 
   //      High warning activation threshold = SP_WRN_H_VAL
   //      High warning reset threshold          = calcHystAbs
   // 
   // Note:    The hysteresis is only checked if warning is being evaluated
   // ▄▄▄▄▄▄▄▄▄▄▄▄▄▄▄▄▄▄▄▄▄▄▄▄▄▄▄▄▄▄▄▄▄▄▄▄▄▄▄▄▄▄▄▄
   RUNG wire#powerrail
      Contact( #wrkWrnHEn )
      wire#w1
      { S7_GenerateENO := "TRUE" } Move(in := #STATIC_DATA.SP_WRN_H_HYST_VAL, out1 => #wrkHyst)
   END_RUNG
   RUNG wire#w1
      { S7_Templates := "SrcType := Real" } LT_Contact(in1 := #STATIC_DATA.SP_WRN_H_HYST_VAL, in2 := 0.0)
      { S7_GenerateENO := "TRUE" } Move(in := 0.0, out1 => #wrkHyst)
   END_RUNG
   RUNG wire#w1
      { S7_Templates := "SrcType := Real"; S7_GenerateENO := "TRUE" } Sub(in1 := #STATIC_DATA.SP_WRN_H_VAL, in2 := #wrkHyst, out => #calcHystAbs)
   END_RUNG
   // the same network as SCL:
   IF #wrkWrnHEn THEN #wrkHyst := #STATIC_DATA.SP_WRN_H_HYST_VAL; END_IF;
   IF #wrkWrnHEn AND (#STATIC_DATA.SP_WRN_H_HYST_VAL < 0.0) THEN #wrkHyst := 0.0; END_IF;
   IF #wrkWrnHEn THEN #calcHystAbs := #STATIC_DATA.SP_WRN_H_VAL - #wrkHyst; END_IF;
END_REGION

REGION Network 29: High warning — Check for activation level and ON-DELAY timer
   // ▀▀▀▀▀▀▀▀▀▀▀▀▀▀▀▀▀▀▀▀▀▀▀▀▀▀▀▀▀▀▀▀▀▀▀▀▀▀▀▀▀▀▀▀
   // If the high warning has been enabled and is not masked and the actual_Value is greater than or 
   // equal to the warning setpoint (SP_WRN_H_VAL), but the warning has not yet been triggered 
   // (msg_Wrn_H = 0) then the ON-DELAY phase is active (the warning timer is counting down).
   // 
   // The timer will begin to count down from the value in TIME_WRN_H_ON_DEL using the 200ms 
   // pulse (it will count down in increments of 0.2s). If the high warning timer is less than or equal to 
   // zero, then the ON-DELAY has expired and the High warning message will become active.
   // 
   // If at any point during the ON-DELAY count down, the actual_Value drops below the activation
   // setpoint (SP_WRN_H_VAL), the timer will be reset to the TIME_WRN_H_ON_DEL value, forcing 
   // the ON-DELAY to start again.
   // ▄▄▄▄▄▄▄▄▄▄▄▄▄▄▄▄▄▄▄▄▄▄▄▄▄▄▄▄▄▄▄▄▄▄▄▄▄▄▄▄▄▄▄▄
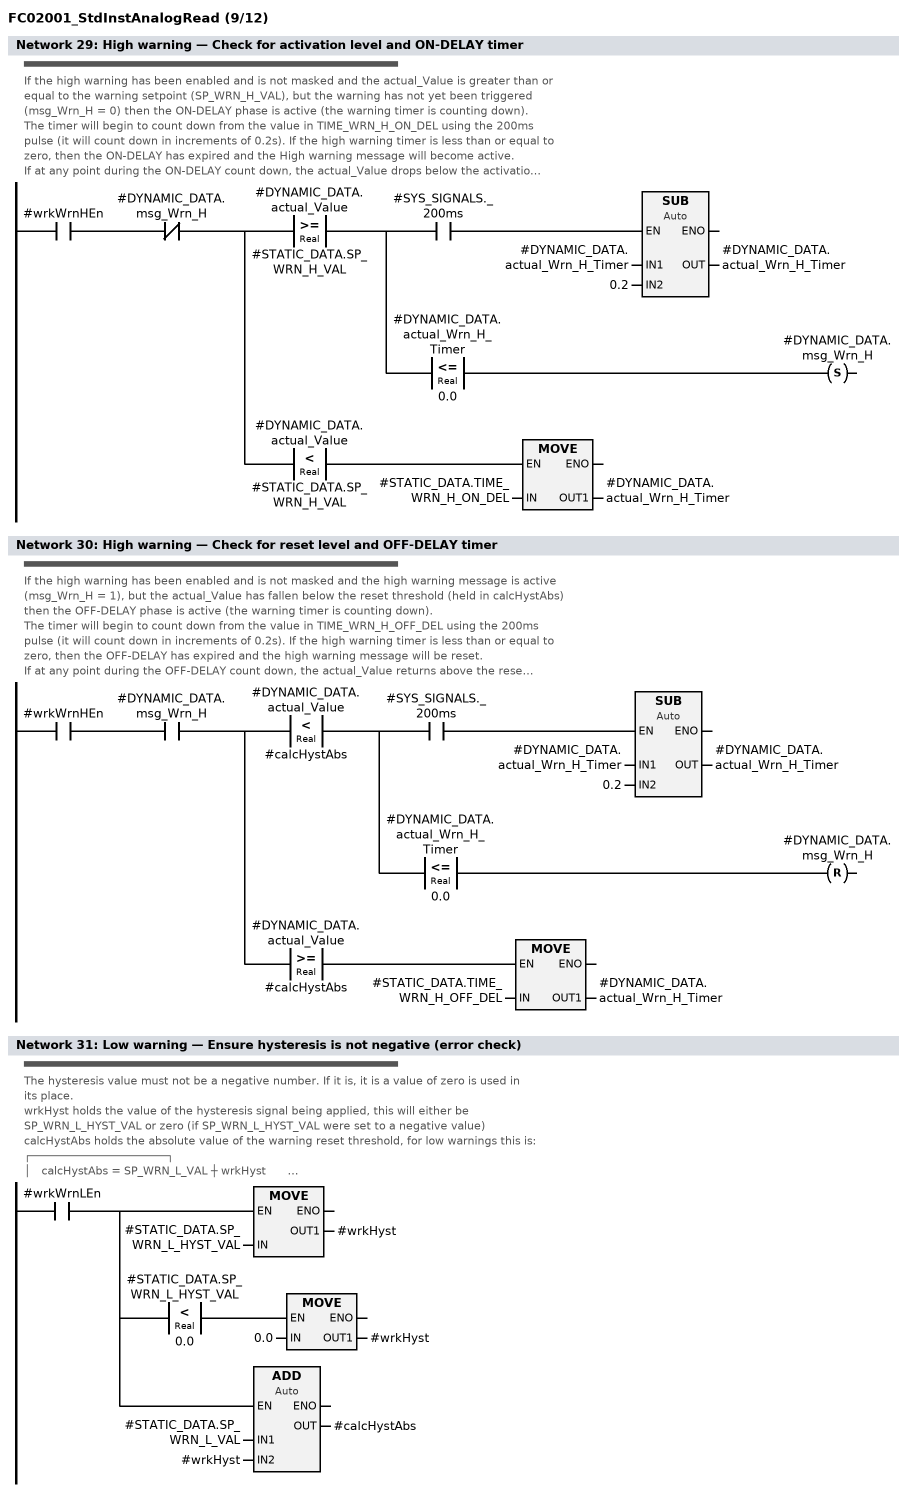
   RUNG wire#powerrail
      Contact( #wrkWrnHEn )
      I_Contact( #DYNAMIC_DATA.msg_Wrn_H )
      wire#w1
      { S7_Templates := "SrcType := Real" } GE_Contact(in1 := #DYNAMIC_DATA.actual_Value, in2 := #STATIC_DATA.SP_WRN_H_VAL)
      wire#w2
      Contact( #SYS_SIGNALS._200ms )
      Sub(in1 := #DYNAMIC_DATA.actual_Wrn_H_Timer, in2 := 0.2, out => #DYNAMIC_DATA.actual_Wrn_H_Timer)
   END_RUNG
   RUNG wire#w2
      { S7_Templates := "SrcType := Real" } LE_Contact(in1 := #DYNAMIC_DATA.actual_Wrn_H_Timer, in2 := 0.0)
      S_Coil( #DYNAMIC_DATA.msg_Wrn_H )
   END_RUNG
   RUNG wire#w1
      { S7_Templates := "SrcType := Real" } LT_Contact(in1 := #DYNAMIC_DATA.actual_Value, in2 := #STATIC_DATA.SP_WRN_H_VAL)
      { S7_GenerateENO := "TRUE" } Move(in := #STATIC_DATA.TIME_WRN_H_ON_DEL, out1 => #DYNAMIC_DATA.actual_Wrn_H_Timer)
   END_RUNG
   // the same network as SCL:
   #_w1 := #wrkWrnHEn AND NOT #DYNAMIC_DATA.msg_Wrn_H;
   #_w2 := #_w1 AND (#DYNAMIC_DATA.actual_Value >= #STATIC_DATA.SP_WRN_H_VAL);
   IF #_w2 AND #SYS_SIGNALS._200ms THEN
       #DYNAMIC_DATA.actual_Wrn_H_Timer := #DYNAMIC_DATA.actual_Wrn_H_Timer - 0.2;
   END_IF;
   IF #_w2 AND (#DYNAMIC_DATA.actual_Wrn_H_Timer <= 0.0) THEN #DYNAMIC_DATA.msg_Wrn_H := TRUE; END_IF;
   IF #_w1 AND (#DYNAMIC_DATA.actual_Value < #STATIC_DATA.SP_WRN_H_VAL) THEN
       #DYNAMIC_DATA.actual_Wrn_H_Timer := #STATIC_DATA.TIME_WRN_H_ON_DEL;
   END_IF;
END_REGION

REGION Network 30: High warning — Check for reset level and OFF-DELAY timer
   // ▀▀▀▀▀▀▀▀▀▀▀▀▀▀▀▀▀▀▀▀▀▀▀▀▀▀▀▀▀▀▀▀▀▀▀▀▀▀▀▀▀▀▀▀
   // If the high warning has been enabled and is not masked and the high warning message is active 
   // (msg_Wrn_H = 1), but the actual_Value has fallen below the reset threshold (held in calcHystAbs) 
   // then the OFF-DELAY phase is active (the warning timer is counting down).
   // 
   // The timer will begin to count down from the value in TIME_WRN_H_OFF_DEL using the 200ms 
   // pulse (it will count down in increments of 0.2s). If the high warning timer is less than or equal to 
   // zero, then the OFF-DELAY has expired and the high warning message will be reset.
   // 
   // If at any point during the OFF-DELAY count down, the actual_Value returns above the reset
   // threshold (calcHystAbs), the timer will be reset to the TIME_WRN_H_OFF_DEL value, forcing 
   // the OFF-DELAY to start again.
   // ▄▄▄▄▄▄▄▄▄▄▄▄▄▄▄▄▄▄▄▄▄▄▄▄▄▄▄▄▄▄▄▄▄▄▄▄▄▄▄▄▄▄▄▄
   RUNG wire#powerrail
      Contact( #wrkWrnHEn )
      Contact( #DYNAMIC_DATA.msg_Wrn_H )
      wire#w1
      { S7_Templates := "SrcType := Real" } LT_Contact(in1 := #DYNAMIC_DATA.actual_Value, in2 := #calcHystAbs)
      wire#w2
      Contact( #SYS_SIGNALS._200ms )
      Sub(in1 := #DYNAMIC_DATA.actual_Wrn_H_Timer, in2 := 0.2, out => #DYNAMIC_DATA.actual_Wrn_H_Timer)
   END_RUNG
   RUNG wire#w2
      { S7_Templates := "SrcType := Real" } LE_Contact(in1 := #DYNAMIC_DATA.actual_Wrn_H_Timer, in2 := 0.0)
      R_Coil( #DYNAMIC_DATA.msg_Wrn_H )
   END_RUNG
   RUNG wire#w1
      { S7_Templates := "SrcType := Real" } GE_Contact(in1 := #DYNAMIC_DATA.actual_Value, in2 := #calcHystAbs)
      { S7_GenerateENO := "TRUE" } Move(in := #STATIC_DATA.TIME_WRN_H_OFF_DEL, out1 => #DYNAMIC_DATA.actual_Wrn_H_Timer)
   END_RUNG
   // the same network as SCL:
   #_w1 := #wrkWrnHEn AND #DYNAMIC_DATA.msg_Wrn_H;
   #_w2 := #_w1 AND (#DYNAMIC_DATA.actual_Value < #calcHystAbs);
   IF #_w2 AND #SYS_SIGNALS._200ms THEN
       #DYNAMIC_DATA.actual_Wrn_H_Timer := #DYNAMIC_DATA.actual_Wrn_H_Timer - 0.2;
   END_IF;
   IF #_w2 AND (#DYNAMIC_DATA.actual_Wrn_H_Timer <= 0.0) THEN #DYNAMIC_DATA.msg_Wrn_H := FALSE; END_IF;
   IF #_w1 AND (#DYNAMIC_DATA.actual_Value >= #calcHystAbs) THEN
       #DYNAMIC_DATA.actual_Wrn_H_Timer := #STATIC_DATA.TIME_WRN_H_OFF_DEL;
   END_IF;
END_REGION

REGION Network 31: Low warning — Ensure hysteresis is not negative (error check)
   // ▀▀▀▀▀▀▀▀▀▀▀▀▀▀▀▀▀▀▀▀▀▀▀▀▀▀▀▀▀▀▀▀▀▀▀▀▀▀▀▀▀▀▀▀
   // The hysteresis value must not be a negative number. If it is, it is a value of zero is used in
   // its place.
   // 
   // wrkHyst holds the value of the hysteresis signal being applied, this will either be 
   // SP_WRN_L_HYST_VAL or zero (if SP_WRN_L_HYST_VAL were set to a negative value)
   // 
   // calcHystAbs holds the absolute value of the warning reset threshold, for low warnings this is:
   // ┌─────────────────────┐
   // │ calcHystAbs = SP_WRN_L_VAL ┼ wrkHyst    │
   // └─────────────────────┘
   // 
   // The two threshold values for the low warning are thus:
   // 
   //      Low warning activation threshold = SP_WRN_L_VAL
   //      Low warning reset threshold          = calcHystAbs
   // 
   // Note:    The hysteresis is only checked if warning is being evaluated
   // ▄▄▄▄▄▄▄▄▄▄▄▄▄▄▄▄▄▄▄▄▄▄▄▄▄▄▄▄▄▄▄▄▄▄▄▄▄▄▄▄▄▄▄▄
   RUNG wire#powerrail
      Contact( #wrkWrnLEn )
      wire#w1
      { S7_GenerateENO := "TRUE" } Move(in := #STATIC_DATA.SP_WRN_L_HYST_VAL, out1 => #wrkHyst)
   END_RUNG
   RUNG wire#w1
      { S7_Templates := "SrcType := Real" } LT_Contact(in1 := #STATIC_DATA.SP_WRN_L_HYST_VAL, in2 := 0.0)
      { S7_GenerateENO := "TRUE" } Move(in := 0.0, out1 => #wrkHyst)
   END_RUNG
   RUNG wire#w1
      Add(in1 := #STATIC_DATA.SP_WRN_L_VAL, in2 := #wrkHyst, out => #calcHystAbs)
   END_RUNG
   // the same network as SCL:
   IF #wrkWrnLEn THEN #wrkHyst := #STATIC_DATA.SP_WRN_L_HYST_VAL; END_IF;
   IF #wrkWrnLEn AND (#STATIC_DATA.SP_WRN_L_HYST_VAL < 0.0) THEN #wrkHyst := 0.0; END_IF;
   IF #wrkWrnLEn THEN #calcHystAbs := #STATIC_DATA.SP_WRN_L_VAL + #wrkHyst; END_IF;
END_REGION

REGION Network 32: Low warning — Check for activation level and ON-DELAY timer
   // ▀▀▀▀▀▀▀▀▀▀▀▀▀▀▀▀▀▀▀▀▀▀▀▀▀▀▀▀▀▀▀▀▀▀▀▀▀▀▀▀▀▀▀▀
   // If the low warning has been enabled and is not masked and the actual_Value is less than or 
   // equal to the warning setpoint (SP_WRN_L_VAL), but the warning has not yet been triggered 
   // (msg_Wrn_L = 0) then the ON-DELAY phase is active (the warning timer is counting down).
   // 
   // The timer will begin to count down from the value in TIME_WRN_L_ON_DEL using the 200ms 
   // pulse (it will count down in increments of 0.2s). If the Low warning timer is less than or equal to 
   // zero, then the ON-DELAY has expired and the Low Warning message will become active.
   // 
   // If at any point during the ON-DELAY count down, the actual_Value rises above the activation
   // setpoint (SP_WRN_L_VAL), the timer will be reset to the TIME_WRN_L_ON_DEL value, forcing 
   // the ON-DELAY to start again.
   // ▄▄▄▄▄▄▄▄▄▄▄▄▄▄▄▄▄▄▄▄▄▄▄▄▄▄▄▄▄▄▄▄▄▄▄▄▄▄▄▄▄▄▄▄
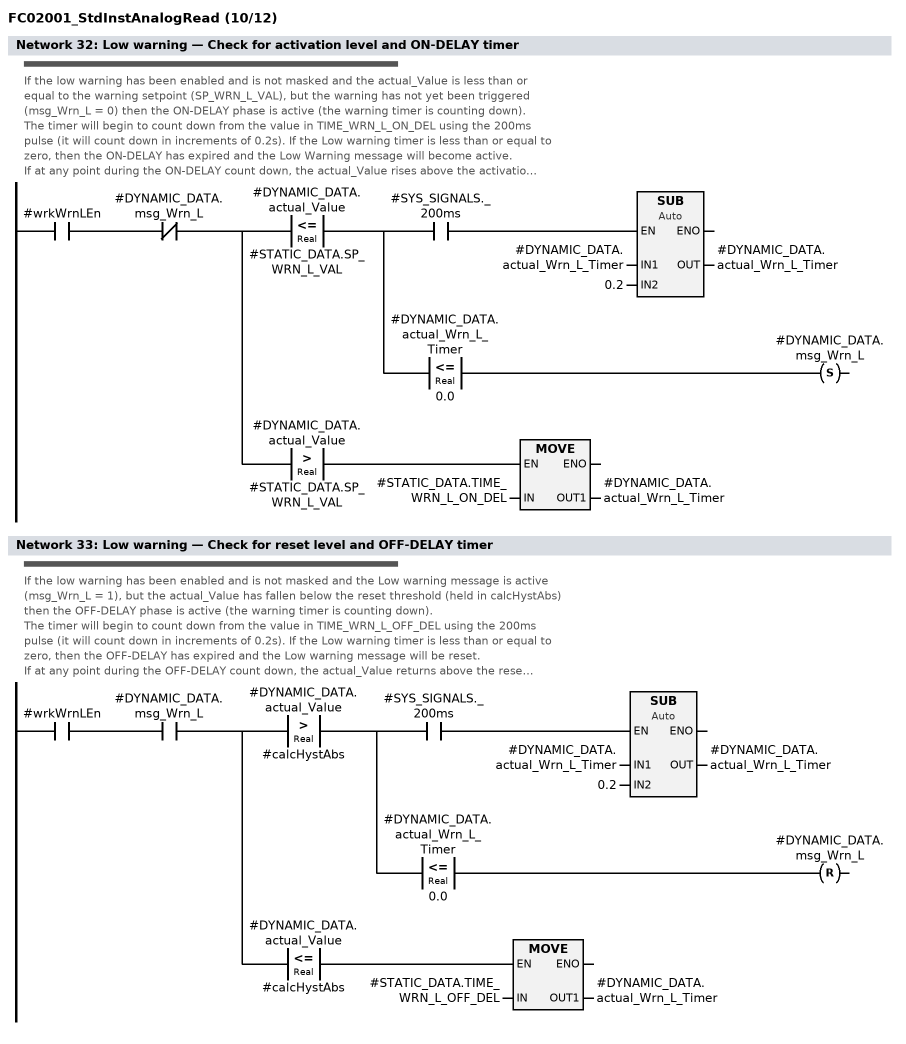
   RUNG wire#powerrail
      Contact( #wrkWrnLEn )
      I_Contact( #DYNAMIC_DATA.msg_Wrn_L )
      wire#w1
      { S7_Templates := "SrcType := Real" } LE_Contact(in1 := #DYNAMIC_DATA.actual_Value, in2 := #STATIC_DATA.SP_WRN_L_VAL)
      wire#w2
      Contact( #SYS_SIGNALS._200ms )
      Sub(in1 := #DYNAMIC_DATA.actual_Wrn_L_Timer, in2 := 0.2, out => #DYNAMIC_DATA.actual_Wrn_L_Timer)
   END_RUNG
   RUNG wire#w2
      { S7_Templates := "SrcType := Real" } LE_Contact(in1 := #DYNAMIC_DATA.actual_Wrn_L_Timer, in2 := 0.0)
      S_Coil( #DYNAMIC_DATA.msg_Wrn_L )
   END_RUNG
   RUNG wire#w1
      { S7_Templates := "SrcType := Real" } GT_Contact(in1 := #DYNAMIC_DATA.actual_Value, in2 := #STATIC_DATA.SP_WRN_L_VAL)
      { S7_GenerateENO := "TRUE" } Move(in := #STATIC_DATA.TIME_WRN_L_ON_DEL, out1 => #DYNAMIC_DATA.actual_Wrn_L_Timer)
   END_RUNG
   // the same network as SCL:
   #_w1 := #wrkWrnLEn AND NOT #DYNAMIC_DATA.msg_Wrn_L;
   #_w2 := #_w1 AND (#DYNAMIC_DATA.actual_Value <= #STATIC_DATA.SP_WRN_L_VAL);
   IF #_w2 AND #SYS_SIGNALS._200ms THEN
       #DYNAMIC_DATA.actual_Wrn_L_Timer := #DYNAMIC_DATA.actual_Wrn_L_Timer - 0.2;
   END_IF;
   IF #_w2 AND (#DYNAMIC_DATA.actual_Wrn_L_Timer <= 0.0) THEN #DYNAMIC_DATA.msg_Wrn_L := TRUE; END_IF;
   IF #_w1 AND (#DYNAMIC_DATA.actual_Value > #STATIC_DATA.SP_WRN_L_VAL) THEN
       #DYNAMIC_DATA.actual_Wrn_L_Timer := #STATIC_DATA.TIME_WRN_L_ON_DEL;
   END_IF;
END_REGION

REGION Network 33: Low warning — Check for reset level and OFF-DELAY timer
   // ▀▀▀▀▀▀▀▀▀▀▀▀▀▀▀▀▀▀▀▀▀▀▀▀▀▀▀▀▀▀▀▀▀▀▀▀▀▀▀▀▀▀▀▀
   // If the low warning has been enabled and is not masked and the Low warning message is active 
   // (msg_Wrn_L = 1), but the actual_Value has fallen below the reset threshold (held in calcHystAbs) 
   // then the OFF-DELAY phase is active (the warning timer is counting down).
   // 
   // The timer will begin to count down from the value in TIME_WRN_L_OFF_DEL using the 200ms 
   // pulse (it will count down in increments of 0.2s). If the Low warning timer is less than or equal to 
   // zero, then the OFF-DELAY has expired and the Low warning message will be reset.
   // 
   // If at any point during the OFF-DELAY count down, the actual_Value returns above the reset
   // threshold (calcHystAbs), the timer will be reset to the TIME_WRN_L_OFF_DEL value, forcing 
   // the OFF-DELAY to start again.
   // ▄▄▄▄▄▄▄▄▄▄▄▄▄▄▄▄▄▄▄▄▄▄▄▄▄▄▄▄▄▄▄▄▄▄▄▄▄▄▄▄▄▄▄▄
   RUNG wire#powerrail
      Contact( #wrkWrnLEn )
      Contact( #DYNAMIC_DATA.msg_Wrn_L )
      wire#w1
      { S7_Templates := "SrcType := Real" } GT_Contact(in1 := #DYNAMIC_DATA.actual_Value, in2 := #calcHystAbs)
      wire#w2
      Contact( #SYS_SIGNALS._200ms )
      Sub(in1 := #DYNAMIC_DATA.actual_Wrn_L_Timer, in2 := 0.2, out => #DYNAMIC_DATA.actual_Wrn_L_Timer)
   END_RUNG
   RUNG wire#w2
      { S7_Templates := "SrcType := Real" } LE_Contact(in1 := #DYNAMIC_DATA.actual_Wrn_L_Timer, in2 := 0.0)
      R_Coil( #DYNAMIC_DATA.msg_Wrn_L )
   END_RUNG
   RUNG wire#w1
      { S7_Templates := "SrcType := Real" } LE_Contact(in1 := #DYNAMIC_DATA.actual_Value, in2 := #calcHystAbs)
      { S7_GenerateENO := "TRUE" } Move(in := #STATIC_DATA.TIME_WRN_L_OFF_DEL, out1 => #DYNAMIC_DATA.actual_Wrn_L_Timer)
   END_RUNG
   // the same network as SCL:
   #_w1 := #wrkWrnLEn AND #DYNAMIC_DATA.msg_Wrn_L;
   #_w2 := #_w1 AND (#DYNAMIC_DATA.actual_Value > #calcHystAbs);
   IF #_w2 AND #SYS_SIGNALS._200ms THEN
       #DYNAMIC_DATA.actual_Wrn_L_Timer := #DYNAMIC_DATA.actual_Wrn_L_Timer - 0.2;
   END_IF;
   IF #_w2 AND (#DYNAMIC_DATA.actual_Wrn_L_Timer <= 0.0) THEN #DYNAMIC_DATA.msg_Wrn_L := FALSE; END_IF;
   IF #_w1 AND (#DYNAMIC_DATA.actual_Value <= #calcHystAbs) THEN
       #DYNAMIC_DATA.actual_Wrn_L_Timer := #STATIC_DATA.TIME_WRN_L_OFF_DEL;
   END_IF;
END_REGION

REGION Network 34: Status signals
   // ▀▀▀▀▀▀▀▀▀▀▀▀▀▀▀▀▀▀▀▀▀▀▀▀▀▀▀▀▀▀▀▀▀▀▀▀▀▀▀▀▀▀▀▀
   // The status signals for faults, alarms and warnings are either duplicates of the message signals 
   // (signals beginning with msg_) or logical combinations of them.
   // 
   // The following is a full list of the status signals:
   // 
   //  ――――――――――――――――――――――――――――――――――――――――――
   //  SIGNAL          FUNCTION            TYPE   DETAILS
   //  ――――――――――――――――――――――――――――――――――――――――――
   //  status_Alm_H       Identical to: msg_Alm_H    Bool    1 = high alm active, 0 = no alm
   // 
   //  status_Alm_L        Identical to: msg_Alm_L       Bool    1 = low alm active, 0 = no alm
   // 
   //  status_Wrn_H       Identical to: msg_Wrn_H    Bool    1 = high wrn active, 0 = no wrn
   // 
   //  status_Wrn_L        Identical to: msg_Wrn_L     Bool    1 = low wrn active, 0 = no wrn
   // 
   //  status_Alm_H_Mask     High alarm is masked        Bool    1 = alm masked, 0 = normal
   // 
   //  status_Alm_L_Mask      Low alarm is masked         Bool    1 = alm masked, 0 = normal
   // 
   //  status_Wrn_H_Mask     High warning is masked       Bool    1 = wrn masked, 0 = normal
   // 
   //  status_Wrn_L_Mask      Low warning is masked        Bool    1 = wrn masked, 0 = normal
   // 
   //  status_Alm_H_Dis         High alarm is disabled       Bool    1 = alm disabled, 0 = normal
   // 
   //  status_Alm_L_Dis          Low alarm is disabled        Bool    1 = alm disabled, 0 = normal
   // 
   //  status_Wrn_H_Dis         High warning is disabled   Bool    1 = wrn disabled, 0 = normal
   // 
   //  status_Wrn_L_Dis          Low warning is disabled       Bool    1 = wrn disabled, 0 = normal
   // 
   //  status_Fault      Indicates any of the msg_Flt    Bool    1 = fault active, 0 = healthy
   //                signals are active:
   //                  msg_Flt_UnderRange
   //                  msg_Flt_OverRange
   //                  msg_Flt_OutOfRange
   //                  msg_Flt_External 
   //                Note: msg_Flt_OutOfRange is already a combination of
   //                           msg_Flt_UnderRange and msg_Flt_OverRange
   // 
   //  status_SimOn      Status simulation mode on     Bool    1 = sim on, 0 = sim off
   // 
   //  status_RemoteOn     Status remote mode on     Bool    1 = rem on, 0 = rem off
   // 
   // 
   //  status_LocalOn      Status local mode on      Bool    1 = loc on, 0 = loc off 
   // 
   //  status_RLOff      Status ALL mode is on           Bool    1 = ALL mode on, 
   //                               0 = ALL mode off
   //  ――――――――――――――――――――――――――――――――――――――――――
   // ▄▄▄▄▄▄▄▄▄▄▄▄▄▄▄▄▄▄▄▄▄▄▄▄▄▄▄▄▄▄▄▄▄▄▄▄▄▄▄▄▄▄▄▄
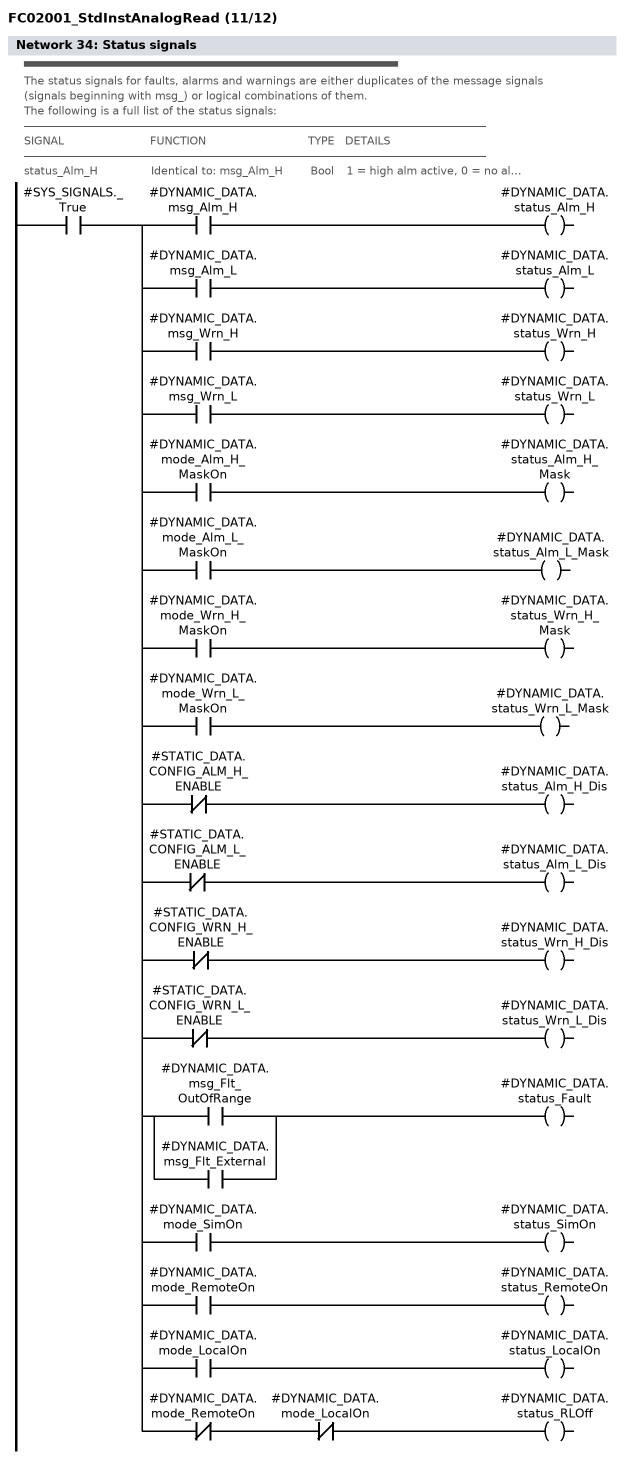
   RUNG wire#powerrail
      Contact( #SYS_SIGNALS._True )
      wire#w1
      Contact( #DYNAMIC_DATA.msg_Alm_H )
      Coil( #DYNAMIC_DATA.status_Alm_H )
   END_RUNG
   RUNG wire#w1
      Contact( #DYNAMIC_DATA.msg_Alm_L )
      Coil( #DYNAMIC_DATA.status_Alm_L )
   END_RUNG
   RUNG wire#w1
      Contact( #DYNAMIC_DATA.msg_Wrn_H )
      Coil( #DYNAMIC_DATA.status_Wrn_H )
   END_RUNG
   RUNG wire#w1
      Contact( #DYNAMIC_DATA.msg_Wrn_L )
      Coil( #DYNAMIC_DATA.status_Wrn_L )
   END_RUNG
   RUNG wire#w1
      Contact( #DYNAMIC_DATA.mode_Alm_H_MaskOn )
      Coil( #DYNAMIC_DATA.status_Alm_H_Mask )
   END_RUNG
   RUNG wire#w1
      Contact( #DYNAMIC_DATA.mode_Alm_L_MaskOn )
      Coil( #DYNAMIC_DATA.status_Alm_L_Mask )
   END_RUNG
   RUNG wire#w1
      Contact( #DYNAMIC_DATA.mode_Wrn_H_MaskOn )
      Coil( #DYNAMIC_DATA.status_Wrn_H_Mask )
   END_RUNG
   RUNG wire#w1
      Contact( #DYNAMIC_DATA.mode_Wrn_L_MaskOn )
      Coil( #DYNAMIC_DATA.status_Wrn_L_Mask )
   END_RUNG
   RUNG wire#w1
      I_Contact( #STATIC_DATA.CONFIG_ALM_H_ENABLE )
      Coil( #DYNAMIC_DATA.status_Alm_H_Dis )
   END_RUNG
   RUNG wire#w1
      I_Contact( #STATIC_DATA.CONFIG_ALM_L_ENABLE )
      Coil( #DYNAMIC_DATA.status_Alm_L_Dis )
   END_RUNG
   RUNG wire#w1
      I_Contact( #STATIC_DATA.CONFIG_WRN_H_ENABLE )
      Coil( #DYNAMIC_DATA.status_Wrn_H_Dis )
   END_RUNG
   RUNG wire#w1
      I_Contact( #STATIC_DATA.CONFIG_WRN_L_ENABLE )
      Coil( #DYNAMIC_DATA.status_Wrn_L_Dis )
   END_RUNG
   RUNG wire#w1
      Contact( #DYNAMIC_DATA.msg_Flt_OutOfRange )
      wire#w2
      Coil( #DYNAMIC_DATA.status_Fault )
   END_RUNG
   RUNG wire#w1
      Contact( #DYNAMIC_DATA.msg_Flt_External )
   END_RUNG wire#w2
   RUNG wire#w1
      Contact( #DYNAMIC_DATA.mode_SimOn )
      Coil( #DYNAMIC_DATA.status_SimOn )
   END_RUNG
   RUNG wire#w1
      Contact( #DYNAMIC_DATA.mode_RemoteOn )
      Coil( #DYNAMIC_DATA.status_RemoteOn )
   END_RUNG
   RUNG wire#w1
      Contact( #DYNAMIC_DATA.mode_LocalOn )
      Coil( #DYNAMIC_DATA.status_LocalOn )
   END_RUNG
   RUNG wire#w1
      I_Contact( #DYNAMIC_DATA.mode_RemoteOn )
      I_Contact( #DYNAMIC_DATA.mode_LocalOn )
      Coil( #DYNAMIC_DATA.status_RLOff )
   END_RUNG
   // the same network as SCL:
   #DYNAMIC_DATA.status_Alm_H := #SYS_SIGNALS._True AND #DYNAMIC_DATA.msg_Alm_H;
   #DYNAMIC_DATA.status_Alm_L := #SYS_SIGNALS._True AND #DYNAMIC_DATA.msg_Alm_L;
   #DYNAMIC_DATA.status_Wrn_H := #SYS_SIGNALS._True AND #DYNAMIC_DATA.msg_Wrn_H;
   #DYNAMIC_DATA.status_Wrn_L := #SYS_SIGNALS._True AND #DYNAMIC_DATA.msg_Wrn_L;
   #DYNAMIC_DATA.status_Alm_H_Mask := #SYS_SIGNALS._True AND #DYNAMIC_DATA.mode_Alm_H_MaskOn;
   #DYNAMIC_DATA.status_Alm_L_Mask := #SYS_SIGNALS._True AND #DYNAMIC_DATA.mode_Alm_L_MaskOn;
   #DYNAMIC_DATA.status_Wrn_H_Mask := #SYS_SIGNALS._True AND #DYNAMIC_DATA.mode_Wrn_H_MaskOn;
   #DYNAMIC_DATA.status_Wrn_L_Mask := #SYS_SIGNALS._True AND #DYNAMIC_DATA.mode_Wrn_L_MaskOn;
   #DYNAMIC_DATA.status_Alm_H_Dis := #SYS_SIGNALS._True AND NOT #STATIC_DATA.CONFIG_ALM_H_ENABLE;
   #DYNAMIC_DATA.status_Alm_L_Dis := #SYS_SIGNALS._True AND NOT #STATIC_DATA.CONFIG_ALM_L_ENABLE;
   #DYNAMIC_DATA.status_Wrn_H_Dis := #SYS_SIGNALS._True AND NOT #STATIC_DATA.CONFIG_WRN_H_ENABLE;
   #DYNAMIC_DATA.status_Wrn_L_Dis := #SYS_SIGNALS._True AND NOT #STATIC_DATA.CONFIG_WRN_L_ENABLE;
   #DYNAMIC_DATA.status_Fault := #SYS_SIGNALS._True AND (#DYNAMIC_DATA.msg_Flt_OutOfRange OR #DYNAMIC_DATA.msg_Flt_External);
   #DYNAMIC_DATA.status_SimOn := #SYS_SIGNALS._True AND #DYNAMIC_DATA.mode_SimOn;
   #DYNAMIC_DATA.status_RemoteOn := #SYS_SIGNALS._True AND #DYNAMIC_DATA.mode_RemoteOn;
   #DYNAMIC_DATA.status_LocalOn := #SYS_SIGNALS._True AND #DYNAMIC_DATA.mode_LocalOn;
   #DYNAMIC_DATA.status_RLOff := #SYS_SIGNALS._True AND NOT #DYNAMIC_DATA.mode_RemoteOn AND NOT #DYNAMIC_DATA.mode_LocalOn;
END_REGION

REGION Network 35: LICENCE AND CONTACT INFORMATION
   // ▀▀▀▀▀▀▀▀▀▀▀▀▀▀▀▀▀▀▀▀▀▀▀▀▀▀▀▀▀▀▀▀▀▀▀▀▀▀▀▀▀▀▀▀
   // LICENCE AND CONTACT INFORMATION
   // 
   // This software and its associated documentation is made available under the MIT Licence:
   // 
   // ════════════════════════════════════════════
   // 
   // The MIT License (MIT)
   // 
   // Copyright © 2020 Michael Gledhill
   // 
   // Permission is hereby granted, free of charge, to any person obtaining a copy of this software 
   // and associated documentation files (the “Software”), to deal in the Software without restriction, 
   // including without limitation the rights to use, copy, modify, merge, publish, distribute, 
   // sublicense, and/or sell copies of the Software, and to permit persons to whom the Software is 
   // furnished to do so, subject to the following conditions: 
   // 
   // The above copyright notice and this permission notice shall be included in all copies or 
   // substantial portions of the Software.
   // 
   // THE SOFTWARE IS PROVIDED “AS IS”, WITHOUT WARRANTY OF ANY KIND, EXPRESS OR IMPLIED, 
   // INCLUDING BUT NOT LIMITED TO THE WARRANTIES OF MERCHANTABILITY, FITNESS FOR A 
   // PARTICULAR PURPOSE AND NON-INFRINGEMENT. IN NO EVENT SHALL THE AUTHORS OR COPYRIGHT 
   // HOLDERS BE LIABLE FOR ANY CLAIM, DAMAGES OR OTHER LIABILITY, WHETHER IN AN ACTION OF 
   // CONTRACT, TORT OR OTHERWISE, ARISING FROM, OUT OF OR IN CONNECTION WITH THE SOFTWARE 
   // OR THE USE OR OTHER DEALINGS IN THE SOFTWARE.
   // 
   // ════════════════════════════════════════════
   //                    ┌────────────┐
   // You can reach the author by email here:   │  mg@practicalseries.com  │
   //                    └────────────┘
   // Questions, corrections, constructive criticism and complaints (polite ones) are invited.
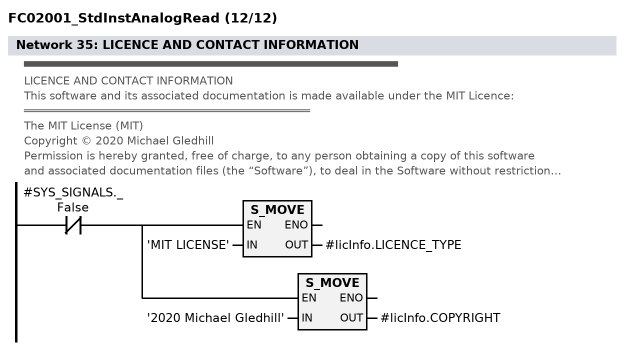
   RUNG wire#powerrail
      I_Contact( #SYS_SIGNALS._False )
      wire#w1
      S_Move(in := 'MIT LICENSE', out => #licInfo.LICENCE_TYPE)
   END_RUNG
   RUNG wire#w1
      S_Move(in := '2020 Michael Gledhill', out => #licInfo.COPYRIGHT)
   END_RUNG
   // the same network as SCL:
   IF NOT #SYS_SIGNALS._False THEN
       #licInfo.LICENCE_TYPE := 'MIT LICENSE';
       #licInfo.COPYRIGHT := '2020 Michael Gledhill';
   END_IF;
END_REGION
END_FUNCTION
